Fanuc KAREL source: ko00080.KL

-- PROVISIONAL review KL for V1013-1; original PC SHA256 3eddf37d0fa57817c33ee1caa3e4ba86973f67b4cd41f306e0b17ca4b0d37c0e
-- Incomplete behavior may be omitted. Consult companion uncertainty JSON. Do not deploy.
PROGRAM KO00080
%NOLOCKGROUP
BEGIN
  -- UNRESOLVED_PC offsets 5-12; opcodes 9D,23
  -- UNRESOLVED_PC offsets 17-66; opcodes 27,22,1C,27,49,7E,AD,22,31,7E,4A
  -- UNRESOLVED_PC offsets 71-75; opcodes 7F
END KO00080
